(* IEC 61131-3 sources: volt/packages/volt-lsp-iec/test-corpus/pro2193/Device/Plc Logic/Application/09 Misc/Library Manager/SysCpuHandling, 11 files *)

(* ---- SYSCPUATOMICADD.pou ---- *)
FUNCTION SYSCPUATOMICADD : DINT
VAR_INPUT
	PIVALUE : POINTER TO DINT;
	NSUM : DINT;
	PRESULT : POINTER TO RTS_IEC_RESULT;
END_VAR
END_FUNCTION

(* ---- SYSCPUATOMICADD64.pou ---- *)
FUNCTION SYSCPUATOMICADD64 : LINT
VAR_INPUT
	PIVALUE : POINTER TO LINT;
	NSUM : LINT;
	PRESULT : POINTER TO RTS_IEC_RESULT;
END_VAR
END_FUNCTION

(* ---- SYSCPUATOMICCOMPAREANDSWAP.pou ---- *)
FUNCTION SYSCPUATOMICCOMPAREANDSWAP : RTS_IEC_RESULT
VAR_INPUT
	PADDRESS : POINTER TO BYTE;
	PSWAPVALUE : POINTER TO BYTE;
	PCOMPAREVALUE : POINTER TO BYTE;
	VALUESIZE : USINT;
END_VAR
END_FUNCTION

(* ---- SYSCPUCALLIECFUNCWITHPARAMS.pou ---- *)
FUNCTION SYSCPUCALLIECFUNCWITHPARAMS : RTS_IEC_RESULT
VAR_INPUT
	PFIECFUNC : POINTER TO BYTE;
	PPARAM : POINTER TO BYTE;
	ULSIZE : UDINT;
END_VAR
END_FUNCTION

(* ---- SYSCPURESETBIT.pou ---- *)
FUNCTION SYSCPURESETBIT : RTS_IEC_RESULT
VAR_INPUT
	PULVALUE : POINTER TO UDINT;
	ULBIT : UDINT;
END_VAR
END_FUNCTION

(* ---- SYSCPURESETBIT2.pou ---- *)
FUNCTION SYSCPURESETBIT2 : RTS_IEC_RESULT
VAR_INPUT
	PBYVALUE : POINTER TO BYTE;
	ULBIT : UDINT;
END_VAR
END_FUNCTION

(* ---- SYSCPUSETBIT.pou ---- *)
FUNCTION SYSCPUSETBIT : RTS_IEC_RESULT
VAR_INPUT
	PULVALUE : POINTER TO UDINT;
	ULBIT : UDINT;
END_VAR
END_FUNCTION

(* ---- SYSCPUSETBIT2.pou ---- *)
FUNCTION SYSCPUSETBIT2 : RTS_IEC_RESULT
VAR_INPUT
	PBYVALUE : POINTER TO BYTE;
	ULBIT : UDINT;
END_VAR
END_FUNCTION

(* ---- SYSCPUTESTANDRESET.pou ---- *)
FUNCTION SYSCPUTESTANDRESET : RTS_IEC_RESULT
VAR_INPUT
	PULVALUE : POINTER TO UDINT;
	ULBIT : UDINT;
END_VAR
END_FUNCTION

(* ---- SYSCPUTESTANDSET.pou ---- *)
FUNCTION SYSCPUTESTANDSET : RTS_IEC_RESULT
VAR_INPUT
	PULVALUE : POINTER TO UDINT;
	ULBIT : UDINT;
END_VAR
END_FUNCTION

(* ---- SYSCPUTESTANDSETBIT.pou ---- *)
FUNCTION SYSCPUTESTANDSETBIT : RTS_IEC_RESULT
VAR_INPUT
	PADDRESS : POINTER TO BYTE;
	NLEN : UDINT;
	IBIT : DINT;
	BSET : DINT;
END_VAR
END_FUNCTION
